// TIA Portal V17 export
// export: Created 2022-08-15T12:23:18.6626076Z, ExportSetting WithDefaults, DisplayName Totally Integrated Automation Portal, DisplayVersion V17, DisplayName TIA Portal Openness, DisplayVersion V17, DisplayName TIA Portal Version Control Interface, DisplayVersion V17, DisplayName SINAMICS Startdrive Advanced, DisplayVersion V17 Update1, DisplayName SINAMICS Startdrive G110M, G120, G120C, G120D, G120P, G115D, DisplayVersion V17 Update1, DisplayName SINAMICS Startdrive G130, G150, S120, S150, SINAMICS MV, S210, DisplayVersion V17 Update1, DisplayName STEP 7 Professional, DisplayVersion V17, DisplayName STEP 7 Safety, DisplayVersion V17, DisplayName WinCC Advanced, DisplayVersion V17
FUNCTION "Routine_3" : Void   // FC3, LAD
{ S7_Optimized_Access := 'TRUE' }
VERSION : 0.1
// stored: AutoNumber true, IsIECCheckEnabled false, SetENOAutomatically false, UDAEnableTagReadback false
BEGIN

REGION Network 1
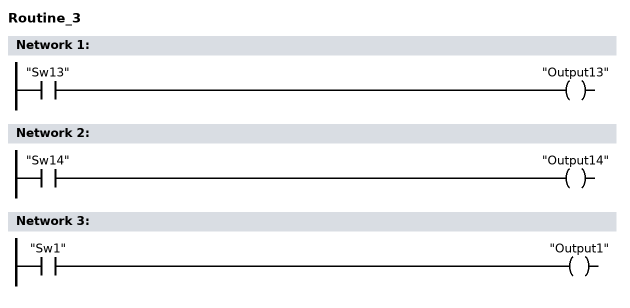
   RUNG wire#powerrail
      Contact( "Sw13" )
      Coil( "Output13" )
   END_RUNG
   // the same network as SCL:
   "Output13" := "Sw13";
END_REGION

REGION Network 2
   RUNG wire#powerrail
      Contact( "Sw14" )
      Coil( "Output14" )
   END_RUNG
   // the same network as SCL:
   "Output14" := "Sw14";
END_REGION

REGION Network 3
   RUNG wire#powerrail
      Contact( "Sw1" )
      Coil( "Output1" )
   END_RUNG
   // the same network as SCL:
   "Output1" := "Sw1";
END_REGION
END_FUNCTION
